TYPE ST_Profile :
(**************************************************************************************
 * 	Application		:	BoxControl Framework
 *	Revision		:	$Revision: 404529 $
 *	Revision date	:	$Date: 2018-04-23 08:21:38 +0200 (Mo., 23 Apr 2018) $
 *	Last changed by	:	$Author: b7bolm $
 *	URL				:	$URL: http://almscdc.swisslog.com/repo/SWPD/Development/BoxControlFramework/20_Release/trunk/01_Software/BCF/BCF/JumpStart/20_Product/10_App/10_Base/10_Lib/10_Conv/01_DUTs/ST_Profile.TcDUT $
 *
 *	Purpose			:	TU Data - Profile
 *
 * ------------------------------------------------------------------------------------
 *	Copyright Swisslog [IP AG], Switzerland. All rights reserved.
 * 
 * ------------------------------------------------------------------------------------
 *	
 * 	Revision History: 
 *
 * 	VERSION			DATE			INITIALS			DESCRIPTION
 *	0.1				01.01.2001		swl					Example
 *
 **************************************************************************************)
STRUCT
	Height			: INT; // Height 
	ProfileLeft		: INT; // Profile left 
	ProfileRight	: INT; // Profile right 
	ProfileFront	: INT; // Profile front 
	ProfileRear		: INT; // Profile rear
	Tunnel			: INT; // Tunnel 
	Runner			: INT; // Runner 
	Weight			: DINT; // Weight 
END_STRUCT
END_TYPE

(* stored: Version 1.1.0.1, ProductVersion 3.1.4022.12
   DUT ST_Profile: Id {65a31a74-7c0e-4f69-8048-7c67241de003} *)
